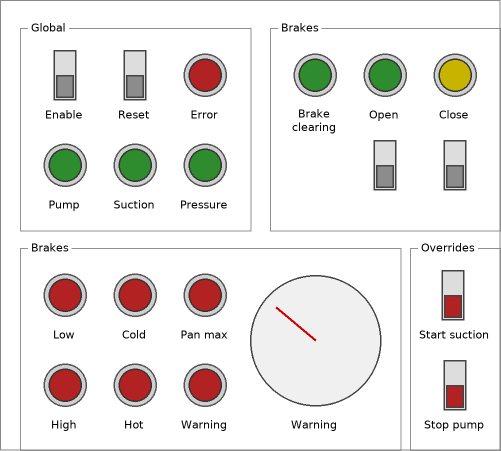
VISUALIZATION Hydraulics  // 501x451
    GroupBox (20,20 231x211), "Global"
        DipSwitch (20,30 50x50), variable: MAIN.HydraulicsControl.bEnable, behaviour: TOGGLE, style: Switch-DipSwitch-Gray
        DipSwitch (90,30 50x50), variable: MAIN.HydraulicsControl.bReset, behaviour: TOGGLE, style: Switch-DipSwitch-Gray
        Lamp1 (160,30 50x50), variable: MAIN.HydraulicsControl.bError, style: Lamp-Lamp1-Red
        Lamp1 (20,120 50x50), variable: MAIN.HydraulicsControl.bPumpRunning, style: Lamp-Lamp1-Green
        Lamp1 (90,120 50x50), variable: MAIN.HydraulicsControl.bSuctionRunning, style: Lamp-Lamp1-Green
        Label (10,80 68x30), "Enable"
        Label (80,80 68x30), "Reset"
        Label (150,80 68x30), "Error"
        Label (10,170 68x30), "Pump"
        Label (80,170 68x30), "Suction"
        Lamp1 (160,120 50x50), variable: MAIN.HydraulicsControl.bOilPressureOK, style: Lamp-Lamp1-Green
        Label (150,170 68x30), "Pressure"
    GroupBox (270,20 231x211), "Brakes"
        DipSwitch (90,120 50x50), variable: MAIN.HydraulicsControl.bOpenBrake, behaviour: TOGGLE, style: Switch-DipSwitch-Gray
        DipSwitch (160,120 50x50), variable: MAIN.HydraulicsControl.bCloseBrake, behaviour: TOGGLE, style: Switch-DipSwitch-Gray
        Lamp1 (160,30 50x50), variable: MAIN.HydraulicsControl.bBrakeClosed, style: Lamp-Lamp1-Yellow
        Lamp1 (20,30 50x50), variable: MAIN.HydraulicsControl.bBrakeClearing, style: Lamp-Lamp1-Green
        Label (150,80 68x30), "Close"
        Label (10,80 68x41), "Brake clearing"
        Lamp1 (90,30 50x50), variable: MAIN.HydraulicsControl.bBrakeOpen, style: Lamp-Lamp1-Green
        Label (80,80 68x30), "Open"
    GroupBox (20,240 381x211), "Brakes"
        Lamp1 (160,30 50x50), variable: MAIN.HydraulicsControl.bOilPanMaximum, style: Lamp-Lamp1-Red
        Label (150,80 68x30), "Pan max"
        Lamp1 (20,30 50x50), variable: MAIN.HydraulicsControl.bOilLow, style: Lamp-Lamp1-Red
        Lamp1 (90,30 50x50), variable: MAIN.HydraulicsControl.bOilCold, style: Lamp-Lamp1-Red
        Label (80,80 68x30), "Cold"
        Label (10,80 68x30), "Low"
        Lamp1 (160,120 50x50), variable: MAIN.HydraulicsControl.bOilWarning, style: Lamp-Lamp1-Red
        Meter360 (230,30 131x141), value: MAIN.HydraulicsControl.fOilLevel, style: Meter-Meter360-Gray, scale format: %.0f, scale 0..120
        Label (260,170 68x30), "Warning"
    Label (170,410 68x30), "Warning"
    Lamp1 (40,360 50x50), variable: MAIN.HydraulicsControl.bOilHigh, style: Lamp-Lamp1-Red
    Lamp1 (110,360 50x50), variable: MAIN.HydraulicsControl.bOilHot, style: Lamp-Lamp1-Red
    Label (100,410 68x30), "Hot"
    Label (30,410 68x30), "High"
    GroupBox (410,240 91x211), "Overrides"
        DipSwitch (18,30 50x50), variable: MAIN.HydraulicsControl.bManualSuction, behaviour: TOGGLE, style: Switch-DipSwitch-Red
        DipSwitch (20,120 50x50), variable: MAIN.HydraulicsControl.bManualPumpStop, behaviour: TOGGLE, style: Switch-DipSwitch-Red
        Label (10,80 68x30), "Start suction"
        Label (10,170 68x30), "Stop pump"
END_VISUALIZATION

(* stored: Version 1.1.0.1, ProductVersion 3.1.4024.15
   Visu Hydraulics: Id {49db7d94-f50f-4256-a167-ca68e51febeb} *)
